// TIA Portal V17 export
// export: Created 2025-03-05T07:58:42.6918127Z, ExportSetting WithDefaults, DisplayName Totally Integrated Automation Portal, DisplayVersion V17 Update 8, DisplayName TIA Portal Openness, DisplayVersion V17 Update 8, DisplayName TIA Portal Version Control Interface, DisplayVersion V17, DisplayName SINAMICS Startdrive Advanced, DisplayVersion V17 SP2, DisplayName SINAMICS Startdrive G110M, G120, G120C, G120D, G120P, G115D, DisplayVersion V17 SP2, DisplayName SINAMICS Startdrive G130, G150, S120, S150, SINAMICS MV, S210, DisplayVersion V17 SP2, DisplayName STEP 7 Professional, DisplayVersion V17 Update 8, DisplayName SINUMERIK ONE STEP 7 Toolbox, DisplayVersion V17 Update 12, DisplayName SINUMERIK 840D sl STEP 7 Toolbox, DisplayVersion V17 Update 12, DisplayName STEP 7 Safety, DisplayVersion V17 Update 6, DisplayName WinCC Advanced, DisplayVersion V17 Update 8
DATA_BLOCK "LBP_AlarmMsgs"   // DB2
TITLE = PLC-Error / Messages / PLC errores/avisos / PLC-Fehler / Meldungen
{ S7_Optimized_Access := 'FALSE'; DB_Accessible_From_OPC_UA := 'FALSE' }
AUTHOR : SINUMERIK
FAMILY : SINUMERIK_ONE
VERSION : 6.15
// Interface between user program and LBP_GenAlarmMsgs [FC10], contains bit arrays for blocking and stop signals as well as fault and status messages. / Interfaz entre programa de usuario y LBP_GenAlarmMsgs [FC10], contiene arrays de bits para bloquear y detener señales, así como avisos de fallo y de estado. / Schnittstelle zwischen Anwenderprogramm und LBP_GenAlarmMsgs [FC10], enthält Bit-Arrays zum Sperren und Stoppen von Signalen sowie Störungs- und Statusmeldungen.
// stored: AutoNumber false, DBAccessibleFromOPCUA false, DBAccessibleFromWebserver true, InstanceOfName LBP_typeAlarmMsgs, InstanceOfType UDT, IsOnlyStoredInLoadMemory false, IsWriteProtectedInAS false
"LBP_typeAlarmMsgs"
   // VAR RETAIN
   //    Chan : Array[1..10] of Struct
   //       FDD : Array[0..15] of Bool;
   //       RID : Array[0..15] of Bool;
   //       NCSD : Array[0..15] of Bool;
   //       FdStop_1 : Array[0..15] of Bool;
   //       FdStop_2 : Array[0..15] of Bool;
   //       FdStop_3 : Array[0..15] of Bool;
   //    END_STRUCT;
   //    Axis : Array[1..31] of Struct
   //       FdStop : Array[0..15] of Bool;
   //    END_STRUCT;
   //    AddValUserA0 : Array[0..63] of Int;
   //    ChanA : Array[1..10] of Struct
   //       FDD_5C00xx : Array[0..15] of Bool;
   //       FDD_RID_5C01xx : Array[0..31] of Bool;
   //       RID_5C02xx : Array[0..31] of Bool;
   //       NCSD_5C03xx : Array[0..15] of Bool;
   //       FdStop_1_5C11xx : Array[0..15] of Bool;
   //       FdStop_2_5C12xx : Array[0..15] of Bool;
   //       FdStop_3_5C13xx : Array[0..15] of Bool;
   //    END_STRUCT;
   //    AxisA : Array[1..31] of Struct
   //       AAFdStop60AAxx : Array[0..15] of Bool;
   //    END_STRUCT;
   //    res552 : Word;
   //    UserA : Array[0..63] of Struct
   //       A70UUxx : Array[0..63] of Bool;
   //    END_STRUCT;
   // END_VAR
BEGIN
END_DATA_BLOCK
